PROGRAM PRG_COM_VLS
VAR
END_VAR

VLS_EP1_CH1_fbSerialLineControl(
    Mode:= SERIALLINEMODE_EL6_22B,
    pComIn:= ADR(VLS_EP1_CH1_stComIn),
    pComOut:=ADR(VLS_EP1_CH1_stComOut),
    SizeComIn:= SIZEOF(VLS_EP1_CH1_stComIn),
    TxBuffer:= VLS_EP1_CH1_SerialTXBuffer,
    RxBuffer:= VLS_EP1_CH1_SerialRXBuffer,
    Error=> ,
    ErrorID=> );

END_PROGRAM

(* stored: Version 1.1.0.1, ProductVersion 3.1.4022.18
   POU PRG_COM_VLS: Id {f650620c-8303-4218-babb-5d1f162a32f7}, SpecialFunc None *)
